{attribute 'enable_dynamic_creation'}	
{attribute 'no_explicit_call' := 'do not call this function block directly'} 
FUNCTION_BLOCK ABSTRACT FileContentTask EXTENDS Task
VAR_INPUT
 	Timeout : TIME := T#2S;
END_VAR
VAR
	_FileContentManager : REFERENCE TO FileContentManager; 
END_VAR

PROPERTY INTERNAL FileContentManager : REFERENCE TO FileContentManager
GET
FileContentManager REF= _FileContentManager;
END_GET
SET
_FileContentManager REF= FileContentManager;
END_SET
END_PROPERTY

METHOD PROTECTED GetErrorMessageByErrorId : WSTRING(255)
VAR_INPUT
	errorId : UDINT;
END_VAR
CASE errorId OF
	1795: GetErrorMessageByErrorId := "invalid or unknown file handle";
	1802: GetErrorMessageByErrorId := "no memory for read buffer";
	1804: GetErrorMessageByErrorId := "file not found";
	1806: GetErrorMessageByErrorId := "file was opened with wrong method";
	1827: GetErrorMessageByErrorId := "folder already exists or invalid sPathName or ePath parameter";
END_CASE

IF GetErrorMessageByErrorId <> "" THEN
	GetErrorMessageByErrorId := WStringHelper.Concat2(": ", GetErrorMessageByErrorId);
END_IF
END_METHOD

METHOD RequestAbort : BOOL
VAR_INPUT
	start : BOOL;
END_VAR
IF Execute(start) = EXECUTION_STATE.BUSY THEN
	RequestAbort := EXECUTION_STATE.BUSY;
ELSE
	RequestAbort := EXECUTION_STATE.DONE;
END_IF
END_METHOD

METHOD PROTECTED Validate
VAR
	//exceptionFactory : ExceptionFactory(__POUNAME(), ClassName, CurrentNamespace.Name);
END_VAR
IF NOT __ISVALIDREF(FileContentManager) THEN
	//exceptionFactory.ThrowException(__POSITION(), "File content menager is not specified");
END_IF

IF FileContentManager.FileHandle = 0 THEN
	//exceptionFactory.ThrowException(__POSITION(), "File is not open");
END_IF
END_METHOD

END_FUNCTION_BLOCK

(* stored: Version 1.1.0.1
   POU FileContentTask: Id {b1426772-2191-466d-91b5-aa0980e0e484}, SpecialFunc None
   Property FileContentManager: Id {95316b75-b424-45bb-97b1-26843b4a2b25}
   Get Get: Id {aab6cba6-f907-4768-b040-7195847efa90}
   Set Set: Id {df151c7c-2c16-43d3-a58c-cad1dfaeee7d}
   Method GetErrorMessageByErrorId: Id {4906c350-513b-4d09-9130-9de049d9da95}
   Method RequestAbort: Id {fa71c439-336d-4f9c-a1c5-d05aade6474d}
   Method Validate: Id {7d61816f-95ff-4e61-86a7-6e2402916cc3} *)
